{attribute 'qualified_only'}
VAR_GLOBAL

// HMI Screen NO
    NowScreen_NO            :    INT    ;       // 현재 화면 위치 NO
	ChangeScreen_NO         :    INT    ;       // PLC 요구 화면 NO

	
// HMI 화면 전환	
	AXIS01					:	BOOL	;
	AXIS02					:	BOOL	;
	AXIS03					:	BOOL	;
	AXIS04					:	BOOL	;
	AXIS05					:	BOOL	;
	
	AXIS01_LAMP				:	BOOL	;
	AXIS02_LAMP				:	BOOL	;
	AXIS03_LAMP				:	BOOL	;
	AXIS04_LAMP				:	BOOL	;
	AXIS05_LAMP				:	BOOL	;
END_VAR

(* stored: Version 1.1.0.1, ProductVersion 3.1.4024.15
   GVL GVL_HMI: Id {7917c9e4-9449-47c7-88e3-a2555ebadac2} *)
